(* Logix 5000 project; controller Good_Foods_96985_10252022_1208 vendor 1 type 14 code 151 rev 32.15; software revision 32.04 *)

TASK MainTask (continuous, watchdog 500 ms) : MainProgram

MODULES
   Local : vendor 1 type 14 code 151 (Compact 0, rev 32.15)
      PLC5103 : 1769-IQ16 (Compact 4, rev 1.1, Input RPI 0.5 ms)
      Analog_IO : Embedded (Compact 2, rev 1.1, Output RPI 80 ms)
      Counters : Embedded (Compact 3, rev 1.1, Output RPI 20 ms)
      Discrete_IO : Embedded (Compact 1, rev 3.1, Output RPI 20 ms)
      DRV3050_RIGHT_AUTOLOAD_CONV_DRV : PowerFlex 525-EENET (Ethernet 192.168.100.11, rev 7.1, Output RPI 20 ms)
      DRV3025_LEFT_AUTOLOAD_CONV_DRV : PowerFlex 525-EENET (Ethernet 192.168.100.10, rev 7.1, Output RPI 20 ms)
      PS2004_Servo_PowerSupply : 2198-P031 (Ethernet 192.168.100.1, rev 11.1, B_MotionSync RPI 2 ms, A_MotionDiagnostics RPI 1 ms)
      DRV2103_ServoDrive01 : vendor 1 type 45 code 10 (Ethernet 192.168.100.2, rev 11.1, B_MotionSync2 RPI 2 ms, A_MotionDiagnostics RPI 1 ms)
END_MODULES

TYPE Container_Recipe :
STRUCT
   sName : STRING;   // Contianer Name
   rLeft_Denester_Park_Pos : REAL;   // Left Denester Park Position
   rRight_Denester_Park_Pos : REAL;   // Right Denester Park Position
   rIndex_Speed : REAL;   // Index Speed
   rLug_Drop_Position : REAL;   // Lug Drop Position
   rSIKO_Rail_Position : REAL;   // SIKO Counter Rail Position
END_STRUCT
END_TYPE

VAR_GLOBAL   (* controller tags *)
   Active_Container_Recipe : Container_Recipe := (sName := 'DELI 12OZ', rLeft_Denester_Park_Pos := 200.0, rRight_Denester_Park_Pos := 96.0, rIndex_Speed := 120.0, rLug_Drop_Position := 40.0, rSIKO_Rail_Position := 99780.0);
   AG_Index_Sys : BOOL := 1;
   Auto_Reset_Timer : TIMER := (PRE := 3000);
   Auto_Reset_Timer2 : TIMER := (PRE := 3500);
   Axis_Virtual_Left_Denest : AXIS_VIRTUAL;
   Axis_Virtual_Right_Denest : AXIS_VIRTUAL;
   bAccess_Allowed : BOOL := 1;
   bAccess_Not_Allowed : BOOL;
   bActive_Cleanout_Mode : BOOL;
   bActive_CleanOut_Mode_Inhibit : BOOL;
   bAll_Doors_OK : BOOL := 1;
   bAll_EStops_OK : BOOL := 1;
   bAlwaysOff : BOOL;
   bAuto_Axis_Reset : BOOL;
   bAuto_Clear_Faults : BOOL;
   bAuto_Disable_Servos : BOOL;
   bAuto_Enable_Servos : BOOL;
   bAuto_Enable_VFDs : BOOL;
   bAuto_Reset_Latch : BOOL;
   bAuto_Reset_Servos : BOOL;
   bbatch_cmd : BOOL;
   bBatch_Cmplt : BOOL;
   bBlink_OFF_250ms : BOOL := 1;
   bBlink_OFF_500ms : BOOL := 1;
   bBlink_ON_250ms : BOOL;
   bBlink_ON_500ms : BOOL := 1;
   bDoor_Safety_Circuit_Active : BOOL;
   bFault_Active : BOOL;
   bFault_Reset_Active : BOOL;
   bHMI_IND_Alarm_Active : BOOL;
   bHMI_IND_Servos_Disable : BOOL;
   bHMI_IND_Servos_Enable : BOOL := 1;
   bHMI_PB_Batch_Count_Reset : BOOL;
   bHMI_PB_Clean_Out : BOOL;
   bHMI_PB_Fault_Reset : BOOL;
   bHMI_PB_Jog_Infeed_Conveyors : BOOL;
   bHMI_PB_JogFwd_Left_Denester : BOOL;
   bHMI_PB_JogFwd_Right_Denester : BOOL;
   bHMI_PB_JogRev_Left_Denester : BOOL;
   bHMI_PB_JogRev_Right_Denester : BOOL;
   bHMI_PB_Left_Denester_Enabled : BOOL := 1;
   bHMI_PB_Left_DropGate_EXT : BOOL;
   bHMI_PB_Left_DropGate_RET : BOOL;
   bHMI_PB_Left_Shuttle_EXT : BOOL;
   bHMI_PB_Left_Shuttle_RET : BOOL;
   bHMI_PB_Load_Recipe : BOOL;
   bHMI_PB_Move_Screws_to_Zero : BOOL;
   bHMI_PB_Park_Denesters : BOOL;
   bHMI_PB_Park_Left_Denester : BOOL;
   bHMI_PB_Park_Right_Denester : BOOL;
   bHMI_PB_Right_Denester_Enabled : BOOL := 1;
   bHMI_PB_Right_DropGate_EXT : BOOL;
   bHMI_PB_Right_DropGate_RET : BOOL;
   bHMI_PB_Right_Shuttle_EXT : BOOL;
   bHMI_PB_Right_Shuttle_RET : BOOL;
   bHMI_PB_Save_Recipe : BOOL;
   bHMI_PB_Servos_Disable : BOOL;
   bHMI_PB_Servos_Enable : BOOL;
   bHmi_PB_Set_Encoder_Home_Position : BOOL;
   bHMI_PB_Start : BOOL;
   bHMI_PB_System_Lifetime_Reset : BOOL;
   bHMI_PB_Teach_Zero_Left_Denester : BOOL;
   bHMI_PB_Teach_Zero_Master_Encoder : BOOL;
   bHMI_PB_Teach_Zero_Right_Denester : BOOL;
   bHMI_PB_Zero_All : BOOL;
   bHome_1 : BOOL;
   bHome_Master_Encoder : BOOL;
   bHoming_Cmplt : BOOL;
   bHoming_Step_1 : BOOL;
   bkDumDum : BOOL;
   bLeft_Denester_Run_Perm : BOOL := 1;
   bLeft_Index_Complete : BOOL;
   bLeft_Index_Cycle_Duration : BOOL := 1;
   bLeft_Indexing : BOOL;
   bLeft_System_Not_Running : BOOL;
   bLeftConvBacklog_OK : BOOL := 1;
   bLeftDropBacklog_OK : BOOL := 1;
   bLeftPrimeBacklog_OK : BOOL := 1;
   bLeftShuttleBacklog_OK : BOOL := 1;
   bMachine_Startup_Delay : BOOL;
   bMaster_Encoder_Homed_After_Restart : BOOL := 1;
   bRight_Denester_Backlog_OK : BOOL;
   bRight_Denester_Run_Perm : BOOL := 1;
   bRight_Index_Complete : BOOL;
   bRight_Index_Cycle_Duration : BOOL := 1;
   bRight_Indexing : BOOL;
   bRight_System_Not_Running : BOOL;
   bRightConvBacklog_OK : BOOL := 1;
   bRightDropBacklog_OK : BOOL := 1;
   bRightPrimeBacklog_OK : BOOL := 1;
   bRightShuttleBacklog_OK : BOOL := 1;
   bSafety_OK : BOOL := 1;
   bScrewsDecoupled : BOOL;
   bSystem_Active : BOOL := 1;
   bSystem_Alarm_Active : BOOL;
   bSystem_Conveyor_Run_Perm : BOOL := 1;
   bSystem_Decouple_CMPLT : BOOL;
   bSystem_Denester_Run_Perm : BOOL := 1;
   bSystem_Gearing_CMPLT : BOOL;
   bSystem_Needs_To_Be_Homed : BOOL;
   bSystem_Park_CMPLT : BOOL;
   bSystem_Sync_CMPLT : BOOL;
   bSystem_VFDStop_CMPLT : BOOL;
   CamP_RampDwn : CAM_PROFILE[40] := ([0].Status := 2, [1].Status := 2, [2].Status := 2, [3].Status := 2);
   CamP_RampUp : CAM_PROFILE[40] := ([0].Status := 2, [1].Status := 2, [2].Status := 2, [3].Status := 2);
   CamP_Run : CAM_PROFILE[40] := ([0].Status := 2, [1].Status := 2);
   Cmplt_Homing_Step_1 : BOOL;
   Container_Recipe : Container_Recipe[32] := ([0].sName := 'CLUB 33OZ', [0].rLeft_Denester_Park_Pos := 280.0, [0].rRight_Denester_Park_Pos := 84.0, [0].rIndex_Speed := 100.0, [0].rLug_Drop_Position := 130.0, [0].rSIKO_Rail_Position := 99695.0, [1].sName := 'CLUB 24 OZ', [1].rLeft_Denester_Park_Pos := 139.0, [1].rRight_Denester_Park_Pos := 322.0, [1].rIndex_Speed := 100.0, [1].rLug_Drop_Position := 200.0, [1].rSIKO_Rail_Position := 99695.0, [2].sName := 'SINGLE SERVE', [2].rLeft_Denester_Park_Pos := 84.0, [2].rRight_Denester_Park_Pos := 280.0, [2].rIndex_Speed := 150.0, [2].rLug_Drop_Position := 240.0, [2].rSIKO_Rail_Position := 99964.0, [3].sName := 'DELI 12OZ', [3].rLeft_Denester_Park_Pos := 200.0, [3].rRight_Denester_Park_Pos := 96.0, [3].rIndex_Speed := 120.0, [3].rLug_Drop_Position := 40.0, [3].rSIKO_Rail_Position := 99780.0, [4].sName := 'DELI 160Z', [4].rLeft_Denester_Park_Pos := 60.0, [4].rRight_Denester_Park_Pos := 290.0, [4].rIndex_Speed := 120.0, [4].rLug_Drop_Position := 20.0, [4].rSIKO_Rail_Position := 99780.0, [5].sName := 'DELI 8OZ', [5].rLeft_Denester_Park_Pos := 345.0, [5].rRight_Denester_Park_Pos := 150.0, [5].rIndex_Speed := 80.0, [5].rLug_Drop_Position := 50.0, [5].rSIKO_Rail_Position := 99780.0);
   ctuBatch_Count : COUNTER := (PRE := 31500, ACC := 3010);
   ctuHour_Count : COUNTER := (PRE := 60);
        .ACC   // Lifetime Counter Rollover 6 month at 90cpm
   ctuInitLeftCyl : COUNTER := (PRE := 1, ACC := 21, DN := 1);
   ctuInitRightCyl : COUNTER := (PRE := 1, ACC := 21, DN := 1);   // Wont Repeat Initilation Sequence If Cmplt
   ctuLeftStartup : COUNTER := (PRE := 4, ACC := 4, DN := 1);
   ctuMinute_Count : COUNTER := (PRE := 60, ACC := 25);
   ctuRightDlyStop : COUNTER := (PRE := 4);
   ctuSecond_Count : COUNTER := (PRE := 60, ACC := 2);
   dAlarms : DINT[8];
        [0].0   // Sync Servos - Timeout Fault
        [0].1   // Gear Servos to Virtuals- Timeout Fault
        [0].10   // Left Drop Gate Not Extended - Timeout Fault
        [0].11   // Containers Not Over Left Drop Gate - Timeout Fault
        [0].12   // Left Drop Gate Retracted - Timeout Fault
        [0].13   // Drop Gate and Shuttle Not In Stop Position - Timeout Fault
        [0].2   // Park Screws - Timeout Fault
        [0].3   // Decouple Screws - Timeout Fault
        [0].4   // Stop VFD's - Timeout Fault
        [0].5   // Container Jam in Front of Right Shuttle
        [0].6   // Right Drop Gate Not Extended - Timeout Fault
        [0].7   // Containers Not Over Right Drop Gate - Timeout Fault
        [0].8   // Right Drop Gate Retracted - Timeout Fault
        [0].9   // Container Jam in Front of Left Shuttle
        [1].0   // HMI Emergency Stop Pressed
        [1].1   // Autoloader Emergency Stop Pressed
        [1].2   // Non Operator Side Emergency Stop Pressed
        [1].3   // Left Operator Side Guard Door Open
        [1].4   // Right Operator Side Guard Door Open
        [1].5   // Left Non Operator Side Guard Door Open
        [1].6   // Right Non Operator Side Guard Door Open
   dHMI_Product_Count : DINT := 63000;
   dHoming_Count : DINT;
   DI_Estop_Autoloader_Pressed : BOOL;
   DI_Estop_HMI_Pressed : BOOL;
   DI_Estop_NonOpSide_Pressed : BOOL;
   DI_PB_Autoloader_Start : BOOL;
   DI_PB_Autoloader_Stop : BOOL := 1;
   DI_PB_Hmi_Jog : BOOL;
   DI_PB_Hmi_Start : BOOL;
   DI_PB_Hmi_Stop : BOOL := 1;
   DI_PE_Left_Conv_Backlog_Present : BOOL := 1;
   DI_PE_Left_Denest_Prime_OK : BOOL := 1;
   DI_PE_Left_Drop_Cont_Present : BOOL := 1;
   DI_PE_Left_Shuttle_Backlog_Present : BOOL := 1;
   DI_PE_Right_Conv_Backlog_Present : BOOL := 1;
   DI_PE_Right_Denest_Prime_OK : BOOL := 1;
   DI_PE_Right_Drop_Cont_Present : BOOL := 1;
   DI_PE_Right_Shuttle_Backlog_Present : BOOL := 1;
   DI_PRX_Left_DropGate_EXT : BOOL;
   DI_PRX_Left_DropGate_RET : BOOL := 1;
   DI_PRX_Left_Shuttle_RET : BOOL := 1;
   DI_PRX_LugChain_HomingProx : BOOL;
   DI_PRX_Right_DropGate_EXT : BOOL;
   DI_PRX_Right_DropGate_RET : BOOL := 1;
   DI_PRX_Right_Shuttle_RET : BOOL := 1;
   DI_PS_Air_Supply_OK : BOOL := 1;
   DI_Safety_Relay_OK : BOOL := 1;
   DI_SS_Left_NonOp_Door_Open : BOOL;
   DI_SS_Left_Op_Door_Open : BOOL;
   DI_SS_Right_NonOp_Door_Open : BOOL;
   DI_SS_Right_Op_Door_Open : BOOL;
   dLeft_Denester_Jog_Dir : DINT := 1;
   dLeft_Shuttle_Seq_CMD : DINT;
   dLeft_Shuttle_Seq_CMPLT : DINT := 3;
        .1   // Retract Left Drop Gate to Drop Containers
        .2   // Extend Left Drop Gate to Accept Containers
        .3   // Extend Left Shuttle to Accept Containers
        .4   // Retract Left Shuttle to move Containers Over Drop Gate
   dMaint_String : DINT;
   dMinute_Count : DINT;
   DO_LT_Stacklight_GRN : BOOL := 1;
   DO_LT_Stacklight_RED : BOOL;
   DO_LT_Stacklight_YLW : BOOL;
   DO_PBLT_Hmi_Reset : BOOL := 1;
   DO_PBLT_Hmi_Start : BOOL := 1;
   DO_SOL_Left_DropGate_EXT : BOOL;
   DO_SOL_Left_DropGate_RET : BOOL;
   DO_SOL_Left_Shuttle_EXT : BOOL;
   DO_SOL_Left_Shuttle_RET : BOOL;
   DO_SOL_Right_DropGate_EXT : BOOL;
   DO_SOL_Right_DropGate_RET : BOOL;
   DO_SOL_Right_Shuttle_EXT : BOOL;
   DO_SOL_Right_Shuttle_RET : BOOL;
   dRight_Denester_Jog_Dir : DINT;
   dRight_Shuttle_Seq_CMD : DINT;
   dRight_Shuttle_Seq_CMPLT : DINT := 3;
        .0   // Right Lane Cylinder Initiliization
        .1   // Retract Right Drop Gate to Drop Containers
        .2   // Extend Right Drop Gate to Accept Containers
        .3   // Extend Right Shuttle to Accept Containers
        .4   // Retract Right Shuttle to move Containers Over Drop Gate
        .5   // System Stopped Release Drop Gate and Retract Shuttle
   dseconds : DINT := 3600;
   dSystem_Lifetime_Count : DINT := 111;
   dSystem_Start_Seq_CMD : DINT;
        .1   // Sync Servos
        .2   // Gear Servos to Lug Belt
   dSystem_Start_Seq_CMPLT : DINT := 6;
        .1   // Sync Servos to Park Position
        .2   // Gear Servos to Virtuals
   dSystem_Stop_Seq_CMD : DINT;
        .1   // Park Screws
        .2   // Decouple Screws
        .3   // Stop VFD's
        .4   // Stop System
   dSystem_Stop_Seq_CMPLT : DINT;
        .0   // Stop Initiated
        .1   // Park Screws
        .2   // Decouple Screws
        .3   // Stop VFD's
        .4   // Stop System
   dTempRevsTime : DINT := 1004;
   Index_Position : INT := 360;
   intHMI_RecipeListPntr : INT := 3;
   intLug_Drop_High_Limit : INT := 45;
   intRecipePntr : INT := 3;
   intStatus_Message : INT := 3;
   Left_Container_Jam_Timer : TIMER := (PRE := 5000);
   Left_Denester : AXIS_CIP_DRIVE;
   Left_Index_Cycle_Duration_Timer : TIMER := (PRE := 1000000000, ACC := 217, EN := 1, TT := 1);
   Left_Index_Measured_Cycle_Time : DINT := 1421;
   Left_Not_Running_Timer : TIMER := (PRE := 4000);
   Left_Rev_Count : INT;
   LugChain_HomingProx_ONS : BOOL;
   LugChain_ONS_Rising : BOOL;
   MAFR_Axis_Virtual : MOTION_INSTRUCTION := (FLAGS := 570425344, DN := 1);
   MAFR_Left_Denester : MOTION_INSTRUCTION := (FLAGS := 536870912, DN := 1, STATE := 1);
   MAFR_Right_Denester : MOTION_INSTRUCTION := (FLAGS := 536870912, DN := 1, STATE := 1);
   MAG_StartGear_LeftDenester : MOTION_INSTRUCTION := (FLAGS := 637534210, DN := 1, IP := 1, DECEL := 1);
   MAG_StartGear_RightDenester : MOTION_INSTRUCTION := (FLAGS := 637534210, DN := 1, IP := 1, DECEL := 1);
   MAH_Axis_Virtual : MOTION_INSTRUCTION := (FLAGS := 704643072, DN := 1, PC := 1, STATE := 17);
   MAH_Left_Denester : MOTION_INSTRUCTION := (FLAGS := 33554432);
   MAH_Master_Encoder : MOTION_INSTRUCTION := (FLAGS := 268435456, ER := 1, ERR := 19);
   MAH_Right_Denester : MOTION_INSTRUCTION := (FLAGS := 33554432);
   MAJ_Left_Denester_Jog : MOTION_INSTRUCTION := (FLAGS := 33554432);
   MAJ_Master_Encoder : MOTION_INSTRUCTION := (FLAGS := 33554432);
   MAJ_Right_Denester_Jog : MOTION_INSTRUCTION := (FLAGS := 33554432);
   MAJ_TEMP_Axis_Master_Follow : MOTION_INSTRUCTION := (FLAGS := 33554432);
   MAM_Home_Left_Denester : MOTION_INSTRUCTION := (FLAGS := 33554432);
   MAM_Home_Right_Denester : MOTION_INSTRUCTION := (FLAGS := 33554432);
   MAM_Left_Denester_Sync : MOTION_INSTRUCTION := (FLAGS := 704643072, DN := 1, PC := 1);
   MAM_Park_Left_Denester : MOTION_INSTRUCTION := (FLAGS := 704643072, DN := 1, PC := 1);
   MAM_Park_Right_Denester : MOTION_INSTRUCTION := (FLAGS := 704643072, DN := 1, PC := 1);
   MAM_Right_Denester_Sync : MOTION_INSTRUCTION := (FLAGS := 704643072, DN := 1, PC := 1);
   mamAxisLeftSCREW_INDEXMOVE : MOTION_INSTRUCTION := (FLAGS := 637534210, DN := 1, IP := 1, DECEL := 1);
   mamAxisRightSCREW_INDEXMOVE : MOTION_INSTRUCTION := (FLAGS := 704643072, DN := 1, PC := 1);
   MAPC_LeftDenesterToLugBelt_RampDwn : MOTION_INSTRUCTION := (FLAGS := 33554432);
   MAPC_LeftDenesterToLugBelt_RampUp : MOTION_INSTRUCTION := (FLAGS := 33554432);
   MAPC_LeftDenesterToLugBelt_Run : MOTION_INSTRUCTION := (FLAGS := 33554432);
   MAPC_RightDenesterToLugBelt_RampDwn : MOTION_INSTRUCTION := (FLAGS := 33554432);
   MAPC_RightDenesterToLugBelt_RampUp : MOTION_INSTRUCTION := (FLAGS := 33554432);
   MAPC_RightDenesterToLugBelt_Run : MOTION_INSTRUCTION := (FLAGS := 33554432);
   MAS_LeftDenester : MOTION_INSTRUCTION := (FLAGS := 704643072, DN := 1, PC := 1);
   MAS_LeftDenester_Jog : MOTION_INSTRUCTION := (FLAGS := 33554432);
   MAS_LeftDenester_Virtual : MOTION_INSTRUCTION := (FLAGS := 704643072, DN := 1, PC := 1);
   MAS_RightDenester : MOTION_INSTRUCTION := (FLAGS := 704643072, DN := 1, PC := 1);
   MAS_RightDenester_Jog : MOTION_INSTRUCTION := (FLAGS := 33554432);
   MAS_RightDenester_Virtual : MOTION_INSTRUCTION := (FLAGS := 704643072, DN := 1, PC := 1);
   MAS_TEMP_Axis_Master_Follow : MOTION_INSTRUCTION := (FLAGS := 704643072, DN := 1, PC := 1);
   MASR_Axis_Virtual : MOTION_INSTRUCTION := (FLAGS := 570425344, DN := 1);
   MASR_Left_Denester : MOTION_INSTRUCTION := (FLAGS := 536870912, DN := 1, STATE := 1);
   MASR_Master_Encoder : MOTION_INSTRUCTION := (FLAGS := 536870912, DN := 1, STATE := 1);
   MASR_Right_Denester : MOTION_INSTRUCTION := (FLAGS := 536870912, DN := 1, STATE := 1);
   Master_Encoder : AXIS_CIP_DRIVE;
   MRP_Axis_Virtual_Sync_Left : MOTION_INSTRUCTION := (FLAGS := 570425344, DN := 1);
   MRP_Axis_Virtual_Sync_Right : MOTION_INSTRUCTION := (FLAGS := 570425344, DN := 1);
   MSF_Left_Denester : MOTION_INSTRUCTION := (FLAGS := 536870912, DN := 1, STATUS := 2, STATE := 1);
   MSF_Right_Denester : MOTION_INSTRUCTION := (FLAGS := 536870912, DN := 1, STATUS := 2, STATE := 1);
   MSO_Left_Denester : MOTION_INSTRUCTION := (FLAGS := 536870912, DN := 1, STATE := 1);
   MSO_Right_Denester : MOTION_INSTRUCTION := (FLAGS := 536870912, DN := 1, STATE := 1);
   ONS : DINT[16] := ([0] := 80);
        [3].0   // HOMING PROX COUNT
        [3].1   // HOMING STEP 1
   OS_System_Inactive : BOOL;
   Power_Supply : AXIS_CIP_DRIVE;
   r_Index_Speed : REAL := 720.0;
   rBatch_Count : REAL := 6020.0;
   rBatch_Count_Both_Lane : REAL := 6020.0;
   rBatch_Count_Pre : REAL := 1.0;
   rConv_Speed : REAL := 9.5;
   rConv_Speed_Hz : DINT := 950;
   rHMI_CleanOut_Time_S : REAL := 120.0;
   rHMI_Drop_Position_Save : REAL := 40.0;
   rHMI_Index_Speed_Save : REAL := 120.0;
   rHMI_Infeed_Conv_Multiplier : REAL := 1.9;
   rHMI_Jog_Speed : REAL := 15.0;
   rHMI_LefPrime_Backlog_Start_Time_S : REAL;
   rHMI_Left_Denester_Park_Pos_Save : REAL := 200.0;
   rHMI_LeftConv_Backlog_Start_Time_S : REAL := 2.0;
   rHMI_LeftConv_Backlog_Stop_Time_S : REAL := 15.0;
   rHMI_LeftDrop_Backlog_Start_Time_S : REAL;
   rHMI_LeftDrop_Backlog_Stop_Time_S : REAL;
   rHMI_LeftPrime_Backlog_Stop_Time_S : REAL;
   rHMI_LeftShuttle_Backlog_Start_Time_S : REAL := 2.0;
   rHMI_LeftShuttle_Backlog_Stop_Time_S : REAL := 2.0;
   rHMI_Machine_Speed : REAL := 5.0;
   rHMI_Right_Denester_Park_Pos_Save : REAL := 96.0;
   rHMI_RightConv_Backlog_Start_Time_S : REAL := 2.0;
   rHMI_RightConv_Backlog_Stop_Time_S : REAL := 15.0;
   rHMI_RightDrop_Backlog_Start_Time_S : REAL;
   rHMI_RightDrop_Backlog_Stop_Time_S : REAL;
   rHMI_RightPrime_Backlog_Start_Time_S : REAL;
   rHMI_RightPrime_Backlog_Stop_Time_S : REAL;
   rHMI_RightShuttle_Backlog_Start_Time_S : REAL;
   rHMI_RightShuttle_Backlog_Stop_Time_S : REAL;
   rHome_Encoder_High_Limit : REAL := 10.0;
   rHome_Encoder_Low_Limit : REAL := 355.0;
   Right_Container_Jam_Timer : TIMER := (PRE := 5000);
   Right_Denester : AXIS_CIP_DRIVE;
   Right_Index_Cycle_Duration_Timer : TIMER := (PRE := 1000000000, ACC := 431, EN := 1, TT := 1);
   Right_Index_Measured_Cycle_Time : DINT := 1421;
   Right_Not_Running_Timer : TIMER := (PRE := 4000);
   Right_Rev_Count : INT;
   Right_System_Running_Timer : TIMER;
   rIndex_Speed_Command : REAL := 280.0;
   rJog_Speed_Command : DINT := 90;
   rLeft_Actual_Throughput : REAL := 42.223785;
   rLeft_Denester_Actual_Position : REAL := 330.16968;
   rLeft_Denester_Position_High : REAL := 12.775666;
   rLeft_Denester_Position_Low : REAL := 10.775666;
   rLug_Conv_Speed_Temp : DINT := 720;
   rMaster_Encoder_Actual_Position : REAL := 84.016;
   rPark_POS_Left_Denester : REAL := 80.0;
   rPark_POS_Right_Denester : REAL;
   rRight_Actual_Throughput : REAL := 42.223785;
   rRight_Denester_Actual_Position : REAL := 268.20654;
   rRight_Denester_Position_High : DINT := 321;
   rRight_Denester_Position_Low : REAL := 224.10654;
   rSIKO_Rail_Position_Save : REAL := 99780.0;
   rSyncHighLimit : REAL := 260.0;
   rSyncLowLimit : REAL := 250.0;
   rSyncPark_Left_Denester : REAL;
   rSyncPark_Right_Denester : REAL;
   rSyncPos_Left_Denester : REAL := 320.0;
   rSyncPos_Right_Denester : REAL := 20.0;
   rSystem_Throughput : REAL := 84.44757;
   rTEMP_Axis_Master_Follow_Actual_Position : REAL;
   rVirtual_Right_Denest_Actual_Position : REAL := 106.68;
   Screw_Accel : REAL := 4000.0;
   Screw_Decel : REAL := 4000.0;
   Servos : MOTION_GROUP;
   strAlarms : STRING[8,32];
   strAlarms_Pre : STRING[8,32] := ([1,0] := 'HMI Emergency Stop Pressed', [1,1] := 'Autoloader Emergency Stop Pressed', [1,2] := 'Non Operator Side Emergency Stop Pressed', [1,3] := 'Left Operator Side Guard Door Open', [1,4] := 'Right Operator Side Guard Door Open', [1,5] := 'Left Non Operator Side Guard Door Open', [1,6] := 'Right Non Operator Side Guard Door Open');
   strEmpty : STRING;
   strEmpty_String : STRING;
   strHMI_Current_User : STRING := 'MAINT';
   String : STRING := 'MAINT';
   strMaint_String : STRING := 'MAINT';
   strMCHS_String : STRING := 'MCHS';
   t1000ms : TIMER := (PRE := 1000, ACC := 877, EN := 1, TT := 1);
   t500ms : TIMER := (PRE := 500, ACC := 105, EN := 1, TT := 1);
   tBatch_Auto_Reset : TIMER := (PRE := 2000);
   tBatch_Dly : TIMER := (PRE := 100);
   tCleanOut : TIMER := (PRE := 120000);
   tDecoupleTimeOut : TIMER := (PRE := 3000);
   TEMP_Axis_Master_Follow : AXIS_VIRTUAL;
   tGearTimeOut : TIMER := (PRE := 3000);
   Timer_AirPressure : TIMER := (PRE := 500);
   tLeftConv_Backlog_Start : TIMER := (PRE := 2000, ACC := 2001, EN := 1, DN := 1);
   tLeftConv_Backlog_Stop : TIMER := (PRE := 15000);
   tLeftDrop_Backlog_Start : TIMER := (ACC := 5, EN := 1, DN := 1);
   tLeftDrop_Backlog_Stop : TIMER;
   tLeftDropGateContTimeOut : TIMER := (PRE := 10000);
   tLeftDropGateExtTimeOut : TIMER := (PRE := 12000);
   tLeftDropGateOpenTimeOut : TIMER := (PRE := 5000);
   tLeftExtDrpDly : TIMER := (PRE := 250);
   tLeftExtShutDly : TIMER := (PRE := 1000);
   tLeftPrime_Backlog_Start : TIMER := (ACC := 2, EN := 1, DN := 1);
   tLeftPrime_Backlog_Stop : TIMER;
   tLeftRetDrpDly : TIMER := (PRE := 250);
   tLeftRetShutDly : TIMER := (PRE := 250);
   tLeftShuttle_Backlog_Start : TIMER := (PRE := 2000, ACC := 2000, EN := 1, DN := 1);
   tLeftShuttle_Backlog_Stop : TIMER := (PRE := 2000);
   tLeftShuttleContPresTimeOut : TIMER := (PRE := 5000);
   tloadconvpress : TIMER := (PRE := 2000);
   tMachine_Startup_Delay : TIMER := (PRE := 20000);
   tParkTimeOut : TIMER := (PRE := 5000);
   tresetdelay : TIMER;
   tRightConv_Backlog_Start : TIMER := (PRE := 2000, ACC := 2000, EN := 1, DN := 1);
   tRightConv_Backlog_Stop : TIMER := (PRE := 15000);
   tRightDrop_Backlog_Start : TIMER := (ACC := 2, EN := 1, DN := 1);
   tRightDrop_Backlog_Stop : TIMER;
   tRightDropGateContTimeOut : TIMER := (PRE := 7000);
   tRightDropGateExtTimeOut : TIMER := (PRE := 12000);
   tRightDropGateOpenTimeOut : TIMER := (PRE := 5000);
   tRightExtDrpDly : TIMER := (PRE := 250);
   tRightExtShutDly : TIMER := (PRE := 1000);
   tRightPrime_Backlog_Start : TIMER := (ACC := 1, EN := 1, DN := 1);
   tRightPrime_Backlog_Stop : TIMER;
   tRightRetDrpDly : TIMER := (PRE := 250);
   tRightRetShutDly : TIMER := (PRE := 250);
   tRightShuttle_Backlog_Start : TIMER := (ACC := 3, EN := 1, DN := 1);
   tRightShuttle_Backlog_Stop : TIMER;
   tRightShuttleContPresTimeOut : TIMER := (PRE := 5000);
   tRightStopPosDly : TIMER := (PRE := 250);
   tRightStopPosTimeOut : TIMER := (PRE := 5000);
   tSafety_Dly_OK : TIMER := (PRE := 5000, ACC := 5002, EN := 1, DN := 1);
   tSecond_Timer : TIMER := (PRE := 1000, ACC := 147, EN := 1, TT := 1);
   tStartUp : TIMER := (PRE := 3000, ACC := 3000, EN := 1, DN := 1);
   tStopVFDsTimeOut : TIMER := (PRE := 5000);
   tSyncTimeOut : TIMER := (PRE := 5000);
   ttempextdly : TIMER := (PRE := 2000);
   tTempRevs : TIMER := (PRE := 999, ACC := 310, EN := 1, TT := 1);
   tTimer_Homing : TIMER := (PRE := 15000);
END_VAR

PROGRAM MainProgram   (* main routine _00_MainRoutine *)
VAR
   intRight_Cycle_Count : INT;
END_VAR

ROUTINE _00_MainRoutine   (* ladder *)
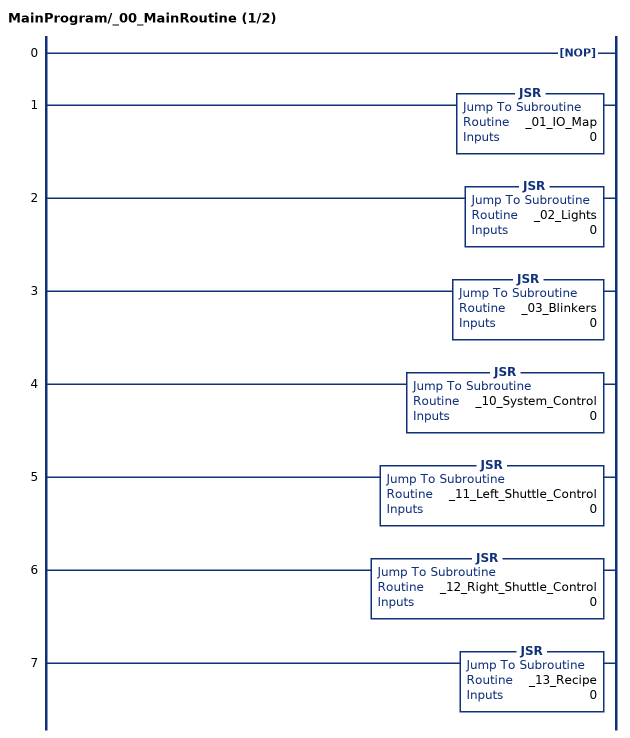
   0: NOP();
   1: JSR(_01_IO_Map,0);
   2: JSR(_02_Lights,0);
   3: JSR(_03_Blinkers,0);
   4: JSR(_10_System_Control,0);
   5: JSR(_11_Left_Shuttle_Control,0);
   6: JSR(_12_Right_Shuttle_Control,0);
   7: JSR(_13_Recipe,0);
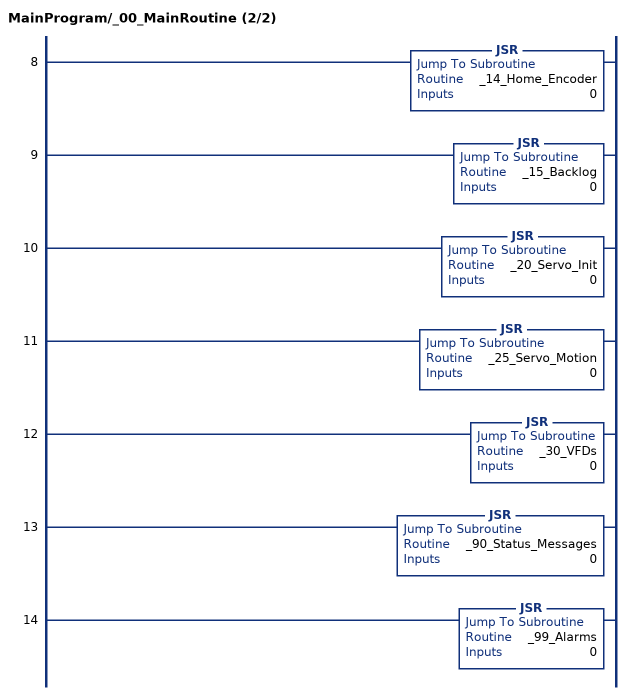
   8: JSR(_14_Home_Encoder,0);
   9: JSR(_15_Backlog,0);
   10: JSR(_20_Servo_Init,0);
   11: JSR(_25_Servo_Motion,0);
   12: JSR(_30_VFDs,0);
   13: JSR(_90_Status_Messages,0);
   14: JSR(_99_Alarms,0);
END_ROUTINE

ROUTINE _01_IO_Map   (* ladder *)
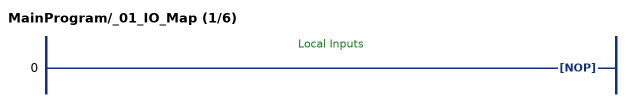
   // Local Inputs
   0: NOP();
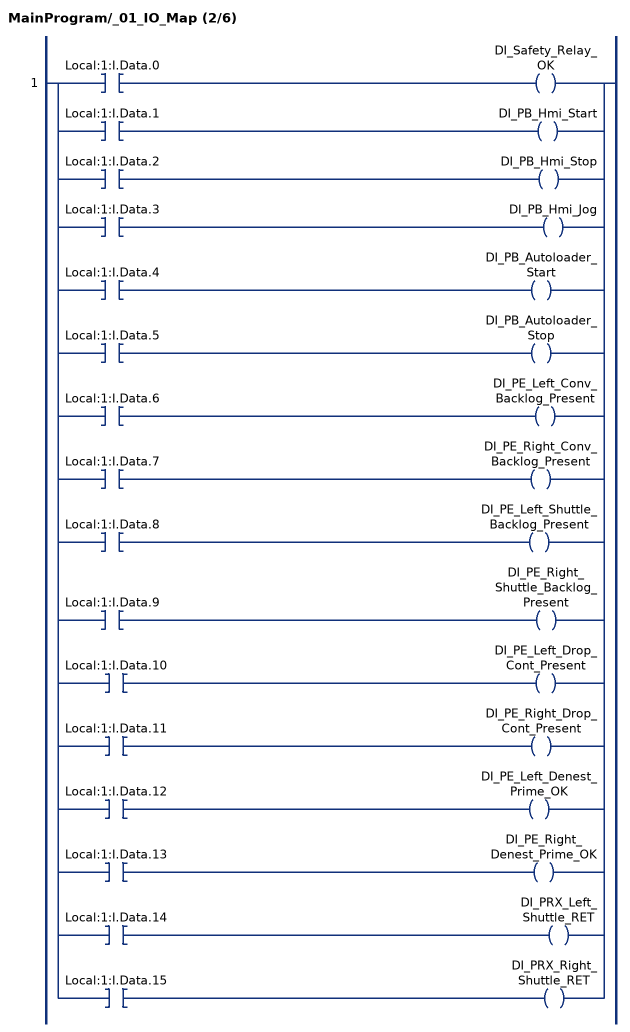
   1: [XIC(Local:1:I.Data.0) OTE(DI_Safety_Relay_OK) ,XIC(Local:1:I.Data.1) OTE(DI_PB_Hmi_Start) ,XIC(Local:1:I.Data.2) OTE(DI_PB_Hmi_Stop) ,XIC(Local:1:I.Data.3) OTE(DI_PB_Hmi_Jog) ,XIC(Local:1:I.Data.4) OTE(DI_PB_Autoloader_Start) ,XIC(Local:1:I.Data.5) OTE(DI_PB_Autoloader_Stop) ,XIC(Local:1:I.Data.6) OTE(DI_PE_Left_Conv_Backlog_Present) ,XIC(Local:1:I.Data.7) OTE(DI_PE_Right_Conv_Backlog_Present) ,XIC(Local:1:I.Data.8) OTE(DI_PE_Left_Shuttle_Backlog_Present) ,XIC(Local:1:I.Data.9) OTE(DI_PE_Right_Shuttle_Backlog_Present) ,XIC(Local:1:I.Data.10) OTE(DI_PE_Left_Drop_Cont_Present) ,XIC(Local:1:I.Data.11) OTE(DI_PE_Right_Drop_Cont_Present) ,XIC(Local:1:I.Data.12) OTE(DI_PE_Left_Denest_Prime_OK) ,XIC(Local:1:I.Data.13) OTE(DI_PE_Right_Denest_Prime_OK) ,XIC(Local:1:I.Data.14) OTE(DI_PRX_Left_Shuttle_RET) ,XIC(Local:1:I.Data.15) OTE(DI_PRX_Right_Shuttle_RET) ];
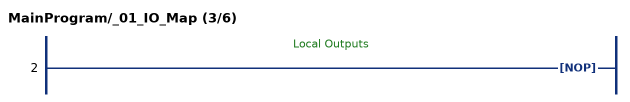
   // Local Outputs
   2: NOP();
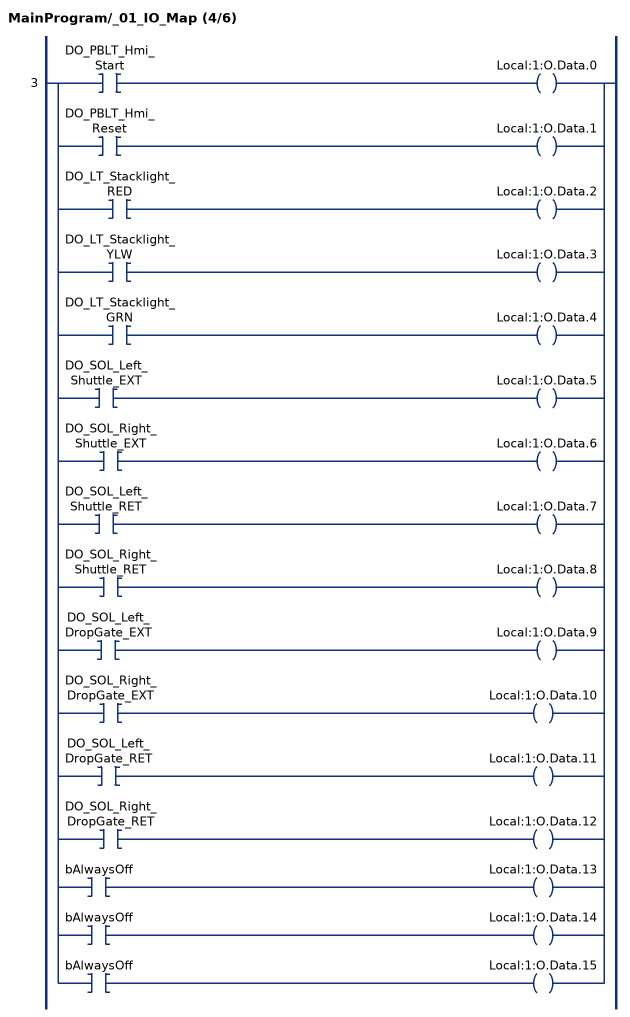
   3: [XIC(DO_PBLT_Hmi_Start) OTE(Local:1:O.Data.0) ,XIC(DO_PBLT_Hmi_Reset) OTE(Local:1:O.Data.1) ,XIC(DO_LT_Stacklight_RED) OTE(Local:1:O.Data.2) ,XIC(DO_LT_Stacklight_YLW) OTE(Local:1:O.Data.3) ,XIC(DO_LT_Stacklight_GRN) OTE(Local:1:O.Data.4) ,XIC(DO_SOL_Left_Shuttle_EXT) OTE(Local:1:O.Data.5) ,XIC(DO_SOL_Right_Shuttle_EXT) OTE(Local:1:O.Data.6) ,XIC(DO_SOL_Left_Shuttle_RET) OTE(Local:1:O.Data.7) ,XIC(DO_SOL_Right_Shuttle_RET) OTE(Local:1:O.Data.8) ,XIC(DO_SOL_Left_DropGate_EXT) OTE(Local:1:O.Data.9) ,XIC(DO_SOL_Right_DropGate_EXT) OTE(Local:1:O.Data.10) ,XIC(DO_SOL_Left_DropGate_RET) OTE(Local:1:O.Data.11) ,XIC(DO_SOL_Right_DropGate_RET) OTE(Local:1:O.Data.12) ,XIC(bAlwaysOff) OTE(Local:1:O.Data.13) ,XIC(bAlwaysOff) OTE(Local:1:O.Data.14) ,XIC(bAlwaysOff) OTE(Local:1:O.Data.15) ];
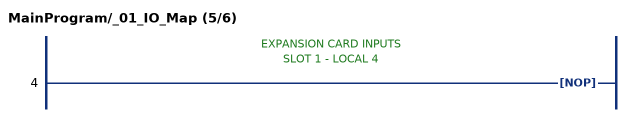
   // EXPANSION CARD INPUTS
   // SLOT 1 - LOCAL 4
   4: NOP();
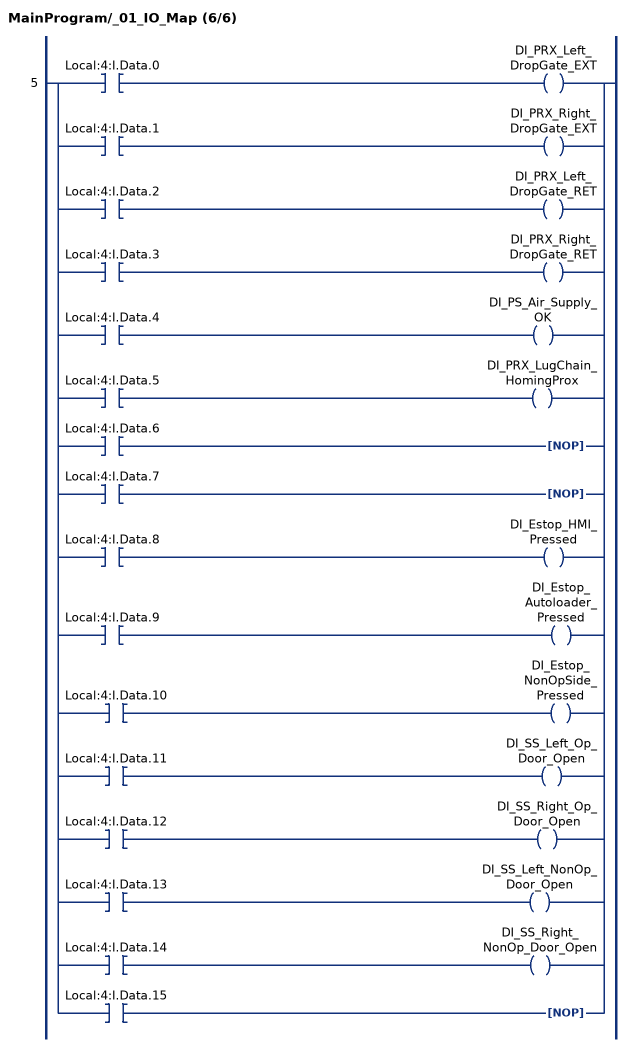
   5: [XIC(Local:4:I.Data.0) OTE(DI_PRX_Left_DropGate_EXT) ,XIC(Local:4:I.Data.1) OTE(DI_PRX_Right_DropGate_EXT) ,XIC(Local:4:I.Data.2) OTE(DI_PRX_Left_DropGate_RET) ,XIC(Local:4:I.Data.3) OTE(DI_PRX_Right_DropGate_RET) ,XIC(Local:4:I.Data.4) OTE(DI_PS_Air_Supply_OK) ,XIC(Local:4:I.Data.5) OTE(DI_PRX_LugChain_HomingProx) ,XIC(Local:4:I.Data.6) NOP() ,XIC(Local:4:I.Data.7) NOP() ,XIC(Local:4:I.Data.8) OTE(DI_Estop_HMI_Pressed) ,XIC(Local:4:I.Data.9) OTE(DI_Estop_Autoloader_Pressed) ,XIC(Local:4:I.Data.10) OTE(DI_Estop_NonOpSide_Pressed) ,XIC(Local:4:I.Data.11) OTE(DI_SS_Left_Op_Door_Open) ,XIC(Local:4:I.Data.12) OTE(DI_SS_Right_Op_Door_Open) ,XIC(Local:4:I.Data.13) OTE(DI_SS_Left_NonOp_Door_Open) ,XIC(Local:4:I.Data.14) OTE(DI_SS_Right_NonOp_Door_Open) ,XIC(Local:4:I.Data.15) NOP() ];
END_ROUTINE

ROUTINE _02_Lights   (* ladder *)
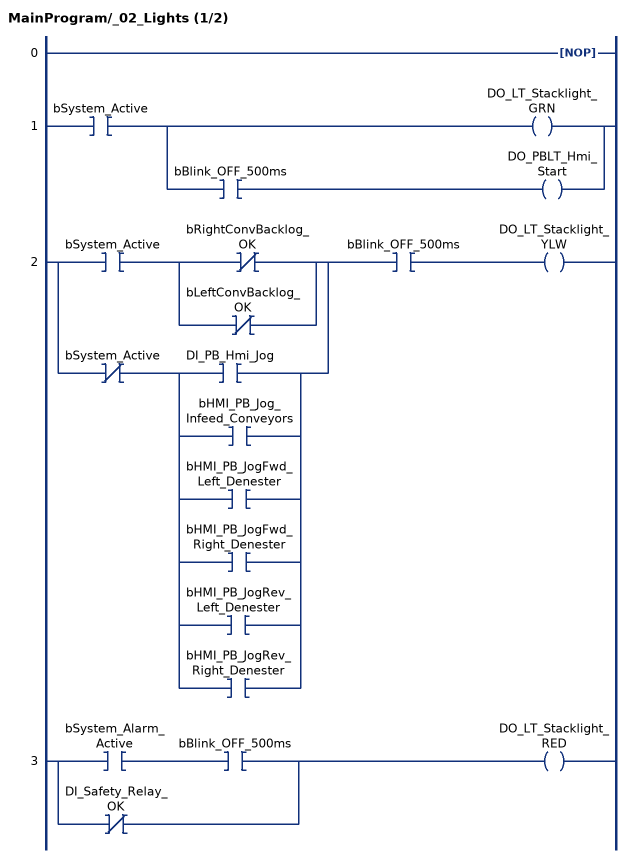
   0: NOP();
   1: XIC(bSystem_Active)[OTE(DO_LT_Stacklight_GRN) ,XIC(bBlink_OFF_500ms) OTE(DO_PBLT_Hmi_Start) ];
   2: [XIC(bSystem_Active) [XIO(bRightConvBacklog_OK) ,XIO(bLeftConvBacklog_OK) ] ,XIO(bSystem_Active) [XIC(DI_PB_Hmi_Jog) ,XIC(bHMI_PB_Jog_Infeed_Conveyors) ,XIC(bHMI_PB_JogFwd_Left_Denester) ,XIC(bHMI_PB_JogFwd_Right_Denester) ,XIC(bHMI_PB_JogRev_Left_Denester) ,XIC(bHMI_PB_JogRev_Right_Denester) ] ]XIC(bBlink_OFF_500ms)OTE(DO_LT_Stacklight_YLW);
   3: [XIC(bSystem_Alarm_Active) XIC(bBlink_OFF_500ms) ,XIO(DI_Safety_Relay_OK) ]OTE(DO_LT_Stacklight_RED);
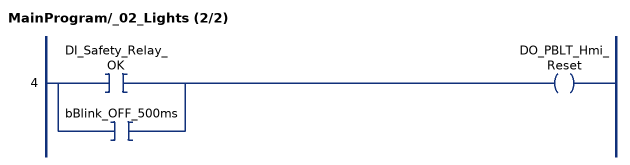
   4: [XIC(DI_Safety_Relay_OK) ,XIC(bBlink_OFF_500ms) ]OTE(DO_PBLT_Hmi_Reset);
END_ROUTINE

ROUTINE _03_Blinkers   (* ladder *)
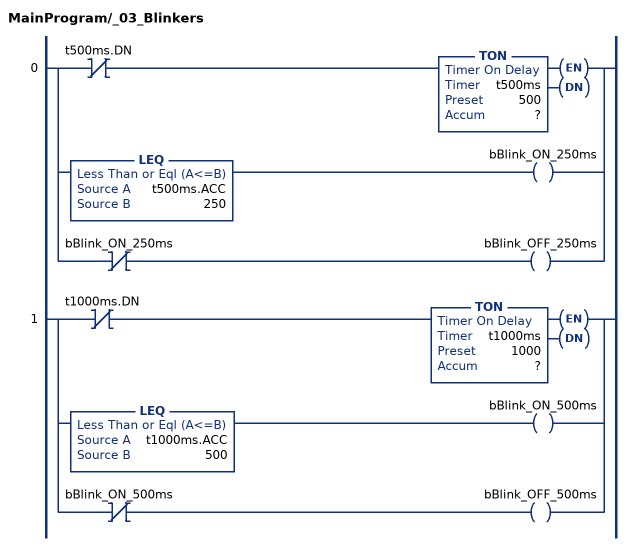
   0: [XIO(t500ms.DN) TON(t500ms,?,?) ,LEQ(t500ms.ACC,250) OTE(bBlink_ON_250ms) ,XIO(bBlink_ON_250ms) OTE(bBlink_OFF_250ms) ];
   1: [XIO(t1000ms.DN) TON(t1000ms,?,?) ,LEQ(t1000ms.ACC,500) OTE(bBlink_ON_500ms) ,XIO(bBlink_ON_500ms) OTE(bBlink_OFF_500ms) ];
END_ROUTINE

ROUTINE _10_System_Control   (* ladder *)
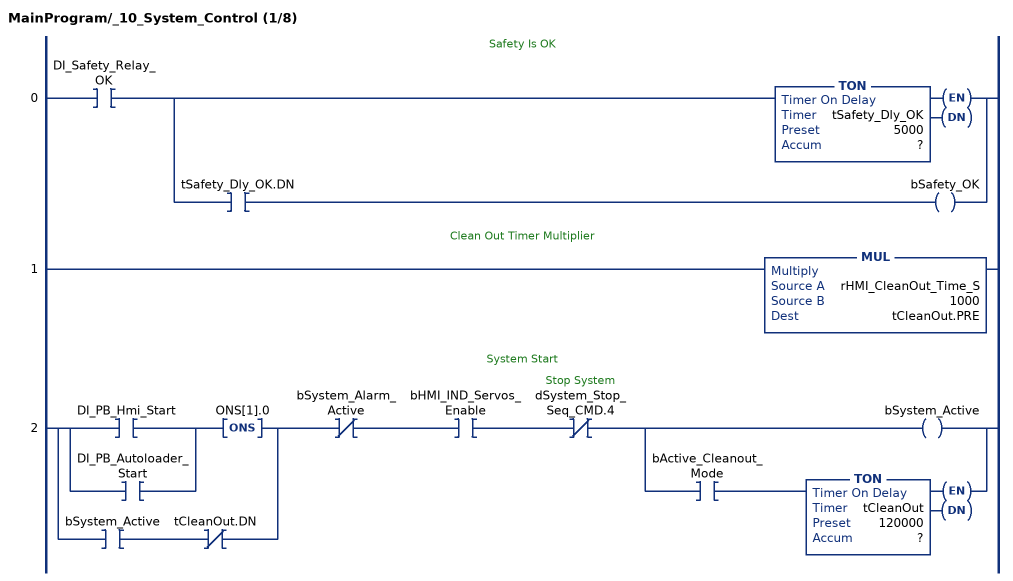
   // Safety Is OK
   0: XIC(DI_Safety_Relay_OK)[TON(tSafety_Dly_OK,?,?) ,XIC(tSafety_Dly_OK.DN) OTE(bSafety_OK) ];
   // Clean Out Timer Multiplier
   1: MUL(rHMI_CleanOut_Time_S,1000,tCleanOut.PRE);
   // System Start
   2: [[XIC(DI_PB_Hmi_Start) ,XIC(DI_PB_Autoloader_Start) ] ONS(ONS[1].0) ,XIC(bSystem_Active) XIO(tCleanOut.DN) ]XIO(bSystem_Alarm_Active)XIC(bHMI_IND_Servos_Enable)XIO(dSystem_Stop_Seq_CMD.4)[OTE(bSystem_Active) ,XIC(bActive_Cleanout_Mode) TON(tCleanOut,?,?) ];
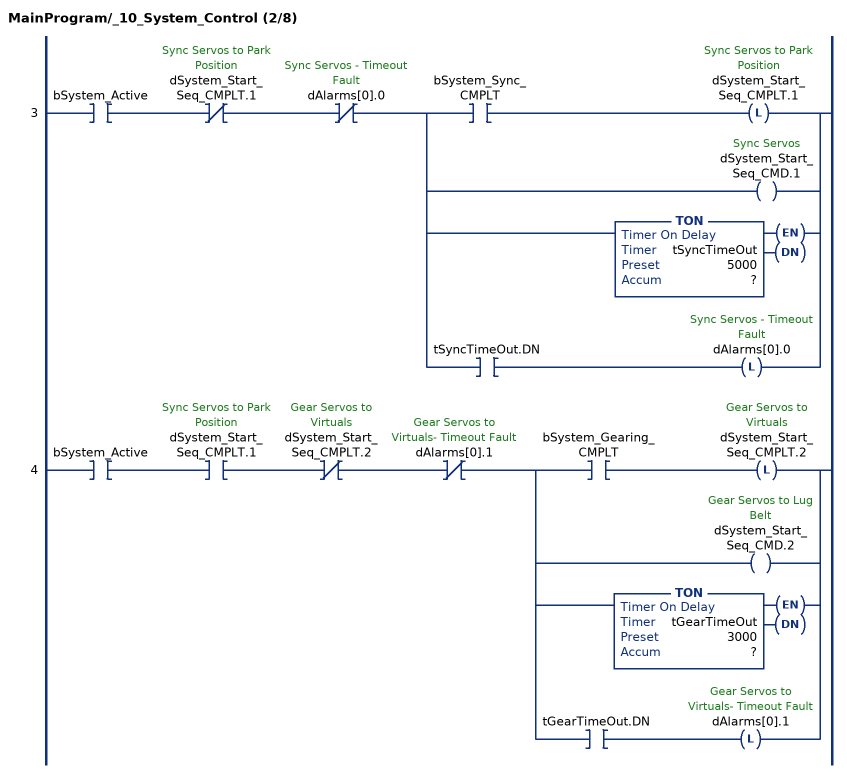
   3: XIC(bSystem_Active)XIO(dSystem_Start_Seq_CMPLT.1)XIO(dAlarms[0].0)[XIC(bSystem_Sync_CMPLT) OTL(dSystem_Start_Seq_CMPLT.1) ,OTE(dSystem_Start_Seq_CMD.1) ,TON(tSyncTimeOut,?,?) ,XIC(tSyncTimeOut.DN) OTL(dAlarms[0].0) ];
   4: XIC(bSystem_Active)XIC(dSystem_Start_Seq_CMPLT.1)XIO(dSystem_Start_Seq_CMPLT.2)XIO(dAlarms[0].1)[XIC(bSystem_Gearing_CMPLT) OTL(dSystem_Start_Seq_CMPLT.2) ,OTE(dSystem_Start_Seq_CMD.2) ,TON(tGearTimeOut,?,?) ,XIC(tGearTimeOut.DN) OTL(dAlarms[0].1) ];
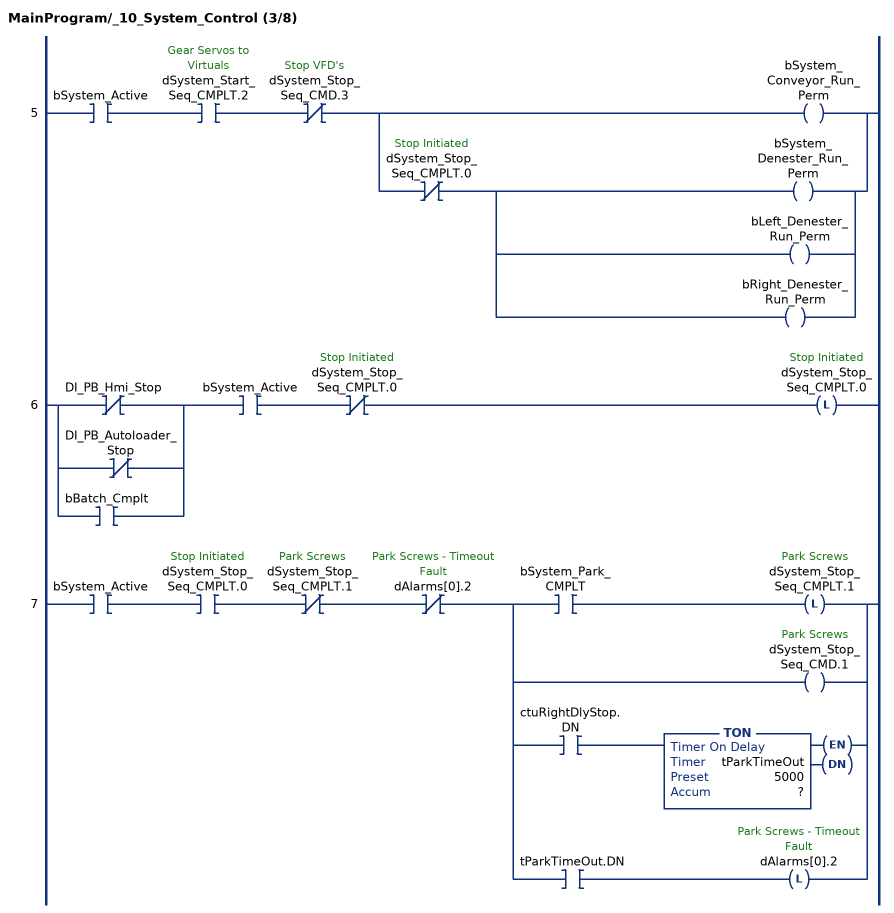
   5: XIC(bSystem_Active)XIC(dSystem_Start_Seq_CMPLT.2)XIO(dSystem_Stop_Seq_CMD.3)[OTE(bSystem_Conveyor_Run_Perm) ,XIO(dSystem_Stop_Seq_CMPLT.0) [OTE(bSystem_Denester_Run_Perm) ,OTE(bLeft_Denester_Run_Perm) ,OTE(bRight_Denester_Run_Perm) ] ];
   6: [XIO(DI_PB_Hmi_Stop) ,XIO(DI_PB_Autoloader_Stop) ,XIC(bBatch_Cmplt) ]XIC(bSystem_Active)XIO(dSystem_Stop_Seq_CMPLT.0)OTL(dSystem_Stop_Seq_CMPLT.0);
   7: XIC(bSystem_Active)XIC(dSystem_Stop_Seq_CMPLT.0)XIO(dSystem_Stop_Seq_CMPLT.1)XIO(dAlarms[0].2)[XIC(bSystem_Park_CMPLT) OTL(dSystem_Stop_Seq_CMPLT.1) ,OTE(dSystem_Stop_Seq_CMD.1) ,XIC(ctuRightDlyStop.DN) TON(tParkTimeOut,?,?) ,XIC(tParkTimeOut.DN) OTL(dAlarms[0].2) ];
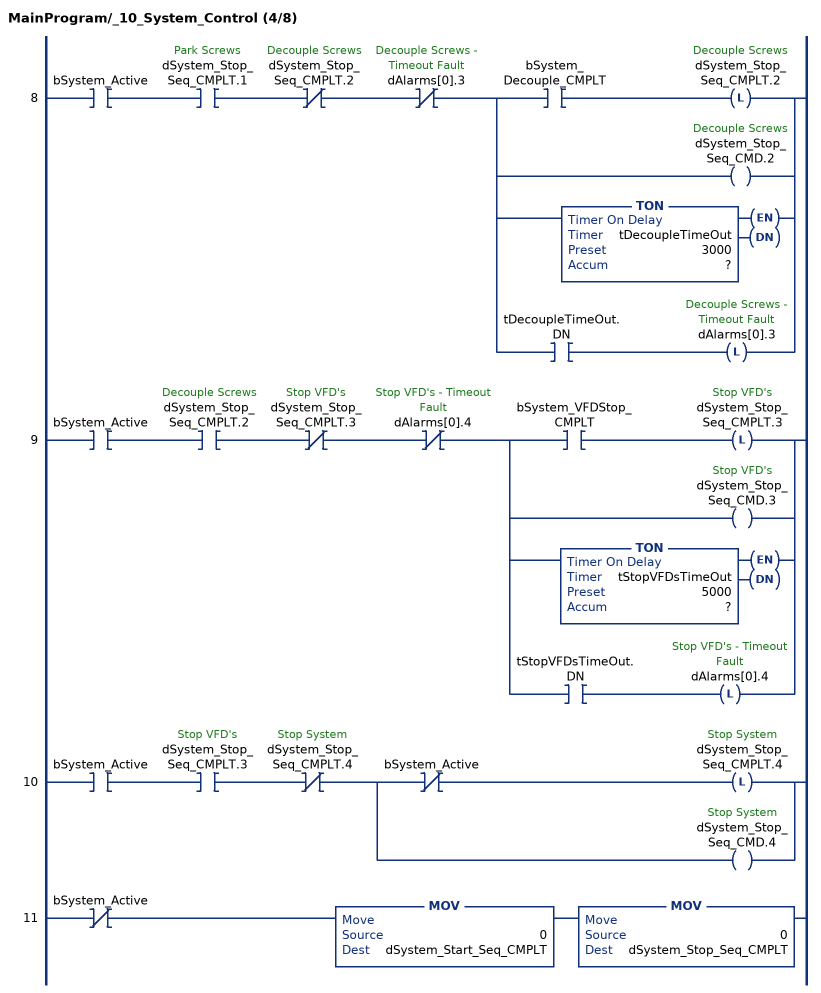
   8: XIC(bSystem_Active)XIC(dSystem_Stop_Seq_CMPLT.1)XIO(dSystem_Stop_Seq_CMPLT.2)XIO(dAlarms[0].3)[XIC(bSystem_Decouple_CMPLT) OTL(dSystem_Stop_Seq_CMPLT.2) ,OTE(dSystem_Stop_Seq_CMD.2) ,TON(tDecoupleTimeOut,?,?) ,XIC(tDecoupleTimeOut.DN) OTL(dAlarms[0].3) ];
   9: XIC(bSystem_Active)XIC(dSystem_Stop_Seq_CMPLT.2)XIO(dSystem_Stop_Seq_CMPLT.3)XIO(dAlarms[0].4)[XIC(bSystem_VFDStop_CMPLT) OTL(dSystem_Stop_Seq_CMPLT.3) ,OTE(dSystem_Stop_Seq_CMD.3) ,TON(tStopVFDsTimeOut,?,?) ,XIC(tStopVFDsTimeOut.DN) OTL(dAlarms[0].4) ];
   10: XIC(bSystem_Active)XIC(dSystem_Stop_Seq_CMPLT.3)XIO(dSystem_Stop_Seq_CMPLT.4)[XIO(bSystem_Active) OTL(dSystem_Stop_Seq_CMPLT.4) ,OTE(dSystem_Stop_Seq_CMD.4) ];
   11: XIO(bSystem_Active)MOV(0,dSystem_Start_Seq_CMPLT)MOV(0,dSystem_Stop_Seq_CMPLT);
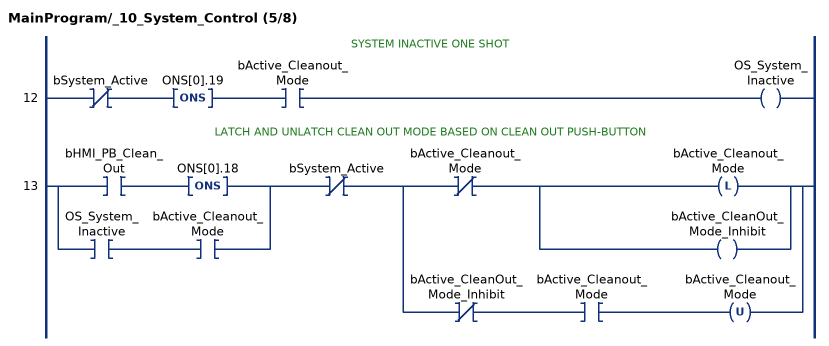
   // SYSTEM INACTIVE ONE SHOT
   12: XIO(bSystem_Active)ONS(ONS[0].19)XIC(bActive_Cleanout_Mode)OTE(OS_System_Inactive);
   // LATCH AND UNLATCH CLEAN OUT MODE BASED ON CLEAN OUT PUSH-BUTTON
   13: [XIC(bHMI_PB_Clean_Out) ONS(ONS[0].18) ,XIC(OS_System_Inactive) XIC(bActive_Cleanout_Mode) ]XIO(bSystem_Active)[XIO(bActive_Cleanout_Mode) [OTL(bActive_Cleanout_Mode) ,OTE(bActive_CleanOut_Mode_Inhibit) ] ,XIO(bActive_CleanOut_Mode_Inhibit) XIC(bActive_Cleanout_Mode) OTU(bActive_Cleanout_Mode) ];
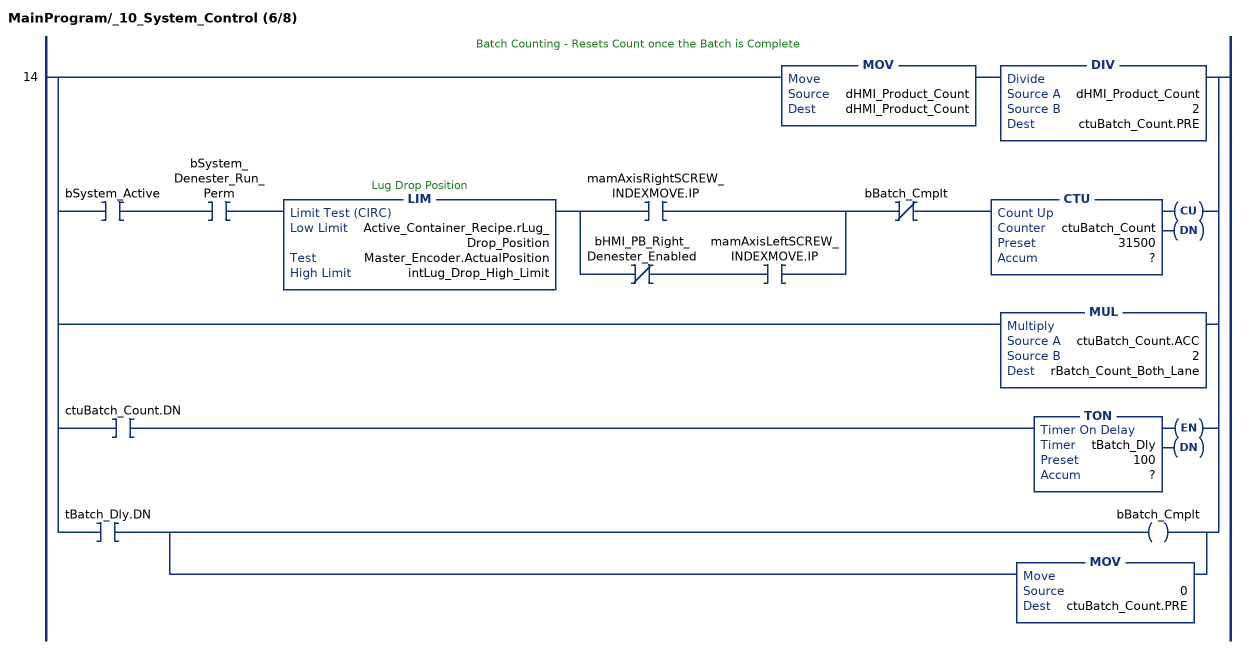
   // Batch Counting - Resets Count once the Batch is Complete
   14: [MOV(dHMI_Product_Count,dHMI_Product_Count) DIV(dHMI_Product_Count,2,ctuBatch_Count.PRE) ,XIC(bSystem_Active) XIC(bSystem_Denester_Run_Perm) LIM(Active_Container_Recipe.rLug_Drop_Position,Master_Encoder.ActualPosition,intLug_Drop_High_Limit) [XIC(mamAxisRightSCREW_INDEXMOVE.IP) ,XIO(bHMI_PB_Right_Denester_Enabled) XIC(mamAxisLeftSCREW_INDEXMOVE.IP) ] XIO(bBatch_Cmplt) CTU(ctuBatch_Count,?,?) ,MUL(ctuBatch_Count.ACC,2,rBatch_Count_Both_Lane) ,XIC(ctuBatch_Count.DN) TON(tBatch_Dly,?,?) ,XIC(tBatch_Dly.DN) [OTE(bBatch_Cmplt) ,MOV(0,ctuBatch_Count.PRE) ] ];
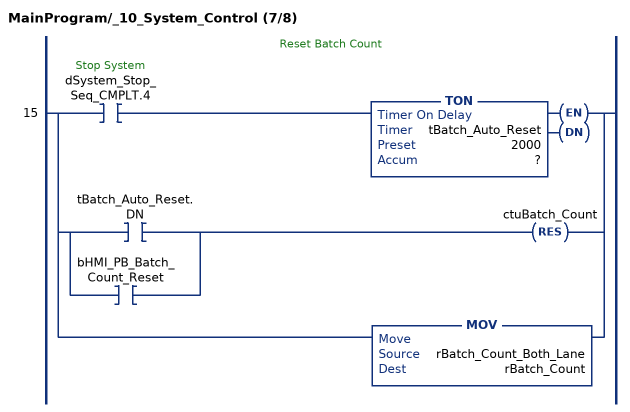
   // Reset Batch Count
   15: [[XIC(dSystem_Stop_Seq_CMPLT.4) TON(tBatch_Auto_Reset,?,?) ,[XIC(tBatch_Auto_Reset.DN) ,XIC(bHMI_PB_Batch_Count_Reset) ] RES(ctuBatch_Count) ] ,MOV(rBatch_Count_Both_Lane,rBatch_Count) ];
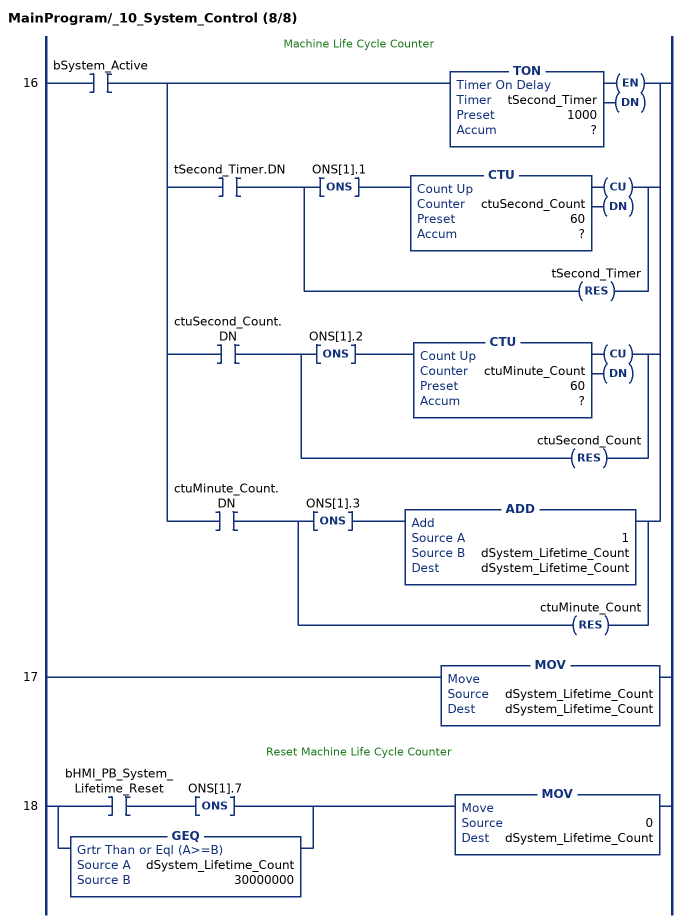
   // Machine Life Cycle Counter
   16: XIC(bSystem_Active)[TON(tSecond_Timer,?,?) ,XIC(tSecond_Timer.DN) [ONS(ONS[1].1) CTU(ctuSecond_Count,?,?) ,RES(tSecond_Timer) ] ,XIC(ctuSecond_Count.DN) [ONS(ONS[1].2) CTU(ctuMinute_Count,?,?) ,RES(ctuSecond_Count) ] ,XIC(ctuMinute_Count.DN) [ONS(ONS[1].3) ADD(1,dSystem_Lifetime_Count,dSystem_Lifetime_Count) ,RES(ctuMinute_Count) ] ];
   17: MOV(dSystem_Lifetime_Count,dSystem_Lifetime_Count);
   // Reset Machine Life Cycle Counter
   18: [XIC(bHMI_PB_System_Lifetime_Reset) ONS(ONS[1].7) ,GEQ(dSystem_Lifetime_Count,30000000) ]MOV(0,dSystem_Lifetime_Count);
END_ROUTINE
